PROGRAM MAIN
VAR
END_VAR

PRG_ProcessSimulation();
PRG_MQTT_Client();

END_PROGRAM

(* stored: Version 1.1.0.1, ProductVersion 3.1.4024.15
   POU MAIN: Id {f559551d-3ebd-43eb-94d2-3d5f7b833ea1}, SpecialFunc None *)
